(* Logix 5000 project; controller Transcat_L33ER vendor 1 type 14 code 107 rev 32.11; software revision 32.02; part 5 of 5 *)
(* tags used below, declared in another part *)
   ActiveRecipe : Recipe;   // Active process recipe downloaded from the HMI recipe system and used by the PLC for automatic operation.
   Device : Device[20];
   RecipeAnyDeviceSelected : BOOL;   // True when at least one device is selected for automatic operation in the active recipe.
   RecipeParametersValid : BOOL;   // True when all selected devices contain valid recipe operating parameters.
   rNum : DINT;   // Index used by RecipeManager to process active recipe device parameters.
   VFD_Panel_Safety_Hoist_1_Cart_OK : ALIAS FOR XS26_VFD_Cabinet_Safety_Controller:I1.Data[2].2;   // HOIST 1 Cart Sensor
   VFD_Panel_Safety_Hoist_2_Cart_OK : ALIAS FOR XS26_VFD_Cabinet_Safety_Controller:I1.Data[2].3;   // HOIST 2 Cart Sensor
(* MainProgram, continued *)

ROUTINE RecipeDeviceLogic   (* ladder *)
// Processes and validates recipe parameters for each device during the RecipeManager FOR loop.
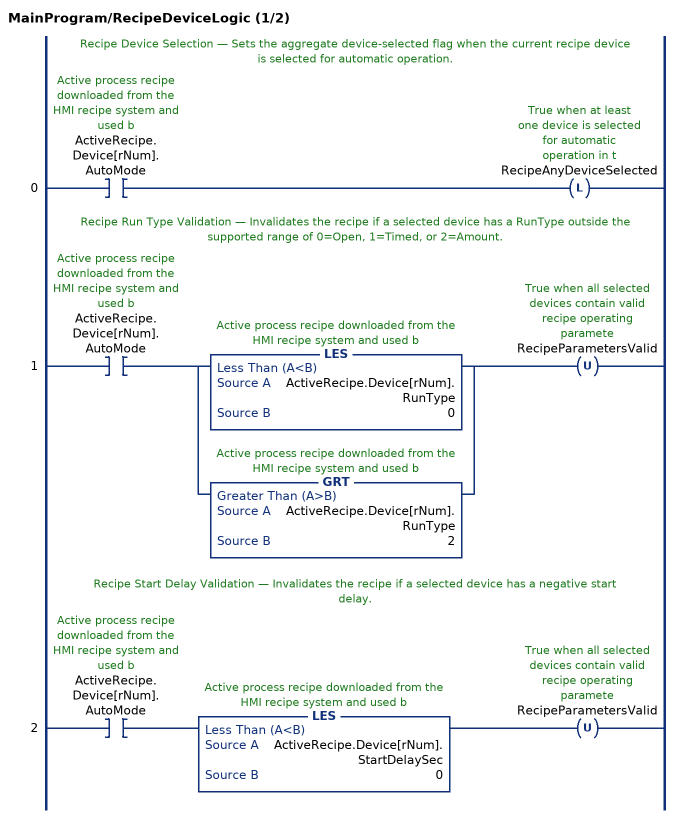
   // Recipe Device Selection — Sets the aggregate device-selected flag when the current recipe device is selected for automatic operation.
   0: XIC(ActiveRecipe.Device[rNum].AutoMode)OTL(RecipeAnyDeviceSelected);
   // Recipe Run Type Validation — Invalidates the recipe if a selected device has a RunType outside the supported range of 0=Open, 1=Timed, or 2=Amount.
   1: XIC(ActiveRecipe.Device[rNum].AutoMode)[LES(ActiveRecipe.Device[rNum].RunType,0) ,GRT(ActiveRecipe.Device[rNum].RunType,2) ]OTU(RecipeParametersValid);
   // Recipe Start Delay Validation — Invalidates the recipe if a selected device has a negative start delay.
   2: XIC(ActiveRecipe.Device[rNum].AutoMode)LES(ActiveRecipe.Device[rNum].StartDelaySec,0)OTU(RecipeParametersValid);
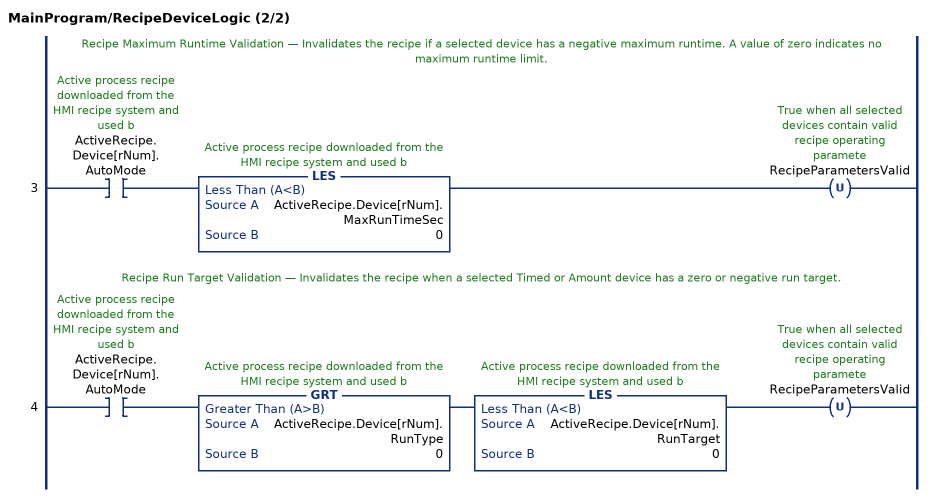
   // Recipe Maximum Runtime Validation — Invalidates the recipe if a selected device has a negative maximum runtime. A value of zero indicates no maximum runtime limit.
   3: XIC(ActiveRecipe.Device[rNum].AutoMode)LES(ActiveRecipe.Device[rNum].MaxRunTimeSec,0)OTU(RecipeParametersValid);
   // Recipe Run Target Validation — Invalidates the recipe when a selected Timed or Amount device has a zero or negative run target.
   4: XIC(ActiveRecipe.Device[rNum].AutoMode)GRT(ActiveRecipe.Device[rNum].RunType,0)LES(ActiveRecipe.Device[rNum].RunTarget,0)OTU(RecipeParametersValid);
END_ROUTINE

ROUTINE RecipeManager   (* ladder *)
// validated and prepares ActiveRecipe
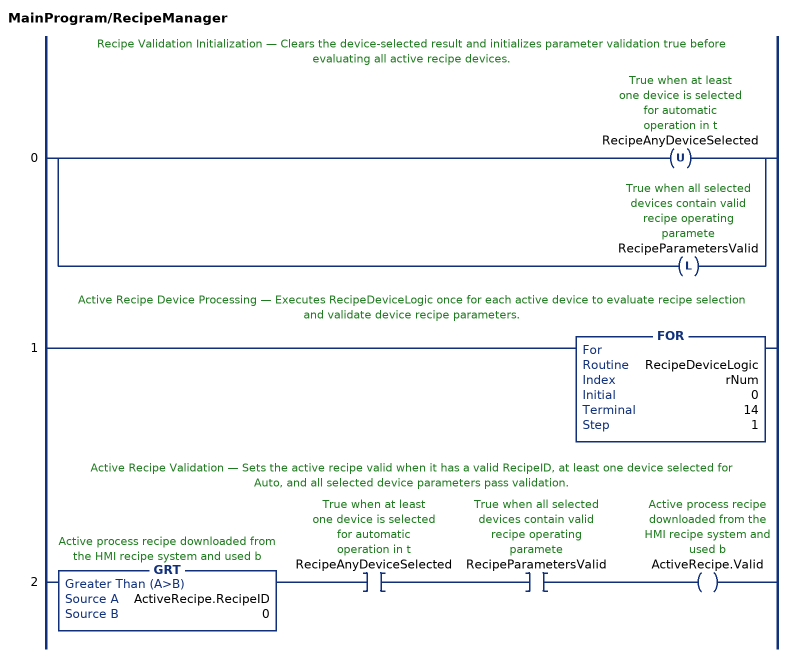
   // Recipe Validation Initialization — Clears the device-selected result and initializes parameter validation true before evaluating all active recipe devices.
   0: [OTU(RecipeAnyDeviceSelected) ,OTL(RecipeParametersValid) ];
   // Active Recipe Device Processing — Executes RecipeDeviceLogic once for each active device to evaluate recipe selection and validate device recipe parameters.
   1: FOR(RecipeDeviceLogic,rNum,0,14,1);
   // Active Recipe Validation — Sets the active recipe valid when it has a valid RecipeID, at least one device selected for Auto, and all selected device parameters pass validation.
   2: GRT(ActiveRecipe.RecipeID,0)XIC(RecipeAnyDeviceSelected)XIC(RecipeParametersValid)OTE(ActiveRecipe.Valid);
END_ROUTINE

ROUTINE Safety_Hoist_Beacons   (* ladder *)
// Saety Hoist Light Beacons
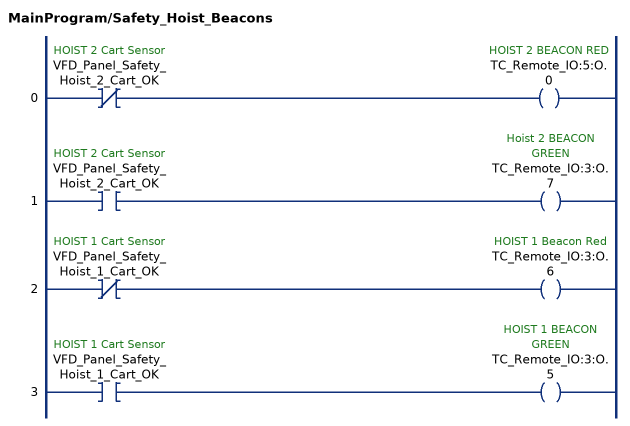
   0: XIO(VFD_Panel_Safety_Hoist_2_Cart_OK)OTE(TC_Remote_IO:5:O.0);
   1: XIC(VFD_Panel_Safety_Hoist_2_Cart_OK)OTE(TC_Remote_IO:3:O.7);
   2: XIO(VFD_Panel_Safety_Hoist_1_Cart_OK)OTE(TC_Remote_IO:3:O.6);
   3: XIC(VFD_Panel_Safety_Hoist_1_Cart_OK)OTE(TC_Remote_IO:3:O.5);
END_ROUTINE
END_PROGRAM
